(* IEC 61131-3 sources: PortalRobot/Portal_robot/Device/application/GVL, 22 files *)

(* ---- GVL_ALARM.gvl.st ---- *)
{attribute 'qualified_only'}
VAR_GLOBAL
	Command : ST_ALARM_COMMAND; // Команды управления журналом аварий
	Status  : ST_ALARM_STATUS; // Сводный статус аварий и предупреждений
	Events  : ARRAY [1..100] OF ST_ALARM_EVENT; // Кольцевой журнал событий
END_VAR

(* ---- GVL_AXIS.gvl.st ---- *)
{attribute 'qualified_only'}
VAR_GLOBAL
	arrAxis : ARRAY [1..3] OF ST_AXIS; // Команды, статусы и диагностика осей X, Y, Z
END_VAR

(* ---- GVL_AXIS_GROUP.gvl.st ---- *)
{attribute 'qualified_only'}
VAR_GLOBAL
	AxisGroup : ST_AXIS_GROUP; // Команды, статусы и диагностика группы XYZ
END_VAR

(* ---- GVL_CELL_CONTROL.gvl.st ---- *)
{attribute 'qualified_only'}
VAR_GLOBAL
	xGlobalError : BOOL; // Глобальная ошибка ячейки
	xReset       : BOOL; // Общий сброс ошибок ячейки
	xManual      : BOOL; // Ручной режим управления ячейкой
	xEnable      : BOOL; // Импульс включения оборудования ячейки
	xDisable     : BOOL; // Импульс отключения оборудования ячейки
	xStart       : BOOL; // Импульс запуска цикла или отмены ожидающей остановки
	xStop        : BOOL; // Импульс остановки автоматического цикла
END_VAR

(* ---- GVL_CELL_MANAGER.gvl.st ---- *)
{attribute 'qualified_only'}
VAR_GLOBAL
	Command : ST_CELL_COMMAND; // Команды менеджера ячейки
	Status  : ST_CELL_STATUS; // Рабочие статусы ячейки
	Diag    : ST_CELL_DIAG; // Состояние автомата ячейки
	Error   : ST_CELL_ERRORS; // Ошибки менеджера ячейки
END_VAR

(* ---- GVL_CELL_SAFETY_IO.gvl.st ---- *)
{attribute 'qualified_only'}
VAR_GLOBAL
	// Логические точки для назначения в Device I/O Mapping. Полярность НЗ-контактов
	// нормализуется при привязке: здесь TRUE всегда означает указанное состояние.
	// Начальное состояние стенда: двери закрыты, грибки отжаты, реле в норме.
	axDoorLockClosedInput : ARRAY [1..4] OF BOOL := [TRUE, TRUE, TRUE, TRUE];
	axDoorUnlockButtonInput : ARRAY [1..4] OF BOOL := [FALSE, FALSE, FALSE, FALSE];
	axEmergencyStopButtonStationInput : ARRAY [1..4] OF BOOL := [FALSE, FALSE, FALSE, FALSE];
	axEmergencyStopCabinetInput : ARRAY [1..2] OF BOOL := [FALSE, FALSE];
	xEmergencyStopMpgInput : BOOL := FALSE;
	xPhaseRelayOkInput    : BOOL := TRUE;
	xPressureRelayOkInput : BOOL := TRUE;
	xSafetyRelayOkInput   : BOOL := TRUE;
	xCellStartButtonInput : BOOL := FALSE;
	xCellStopButtonInput  : BOOL := FALSE;
	xCellResetButtonInput : BOOL := FALSE;
	xMpgAxisXInput : BOOL := FALSE;
	xMpgAxisYInput : BOOL := FALSE;
	xMpgAxisZInput : BOOL := FALSE;
	xMpgMultiplier1Input : BOOL := FALSE;
	xMpgMultiplier10Input : BOOL := FALSE;
	xMpgMultiplier100Input : BOOL := FALSE;

	// Выходы для назначения на физические каналы.
	axDoorUnlockOutput : ARRAY [1..4] OF BOOL;
	axDoorButtonLampOutput : ARRAY [1..4] OF BOOL;
	xSafetyRelayResetOutput : BOOL;
	// Светосигнальная колонна: готовые уровни с миганием из PLC_PRG.RunSignalTower.
	xSignalTowerRedOutput   : BOOL;
	xSignalTowerAmberOutput : BOOL;
	xSignalTowerGreenOutput : BOOL;
END_VAR

(* ---- GVL_CELL_SETTINGS.gvl.st ---- *)
{attribute 'qualified_only'}
VAR_GLOBAL CONSTANT
	// Максимальное число слотов магазина, используемое в статических границах массивов.
	NumberDetail : SINT := 70; // Максимальное число слотов магазина
END_VAR

VAR_GLOBAL
	//Порядок команд для смены, загрузки и выгрузки станков
	CHANGE_MACHINE : ARRAY [0..40] OF ST_MACHINE_RECIPE // Рецепт смены детали в станке
	:=[
	   (eCommand := E_MACHINE_STATE.DOOR_OPEN),
	   (eCommand := E_MACHINE_STATE.ROBOT_ACTION, eRobotAction := E_ROBOT_ACTION.ROTATE_TO_DETAIL),
	   (eCommand := E_MACHINE_STATE.ROBOT_ACTION, eRobotAction := E_ROBOT_ACTION.UNCLAMP_2),
	   (eCommand := E_MACHINE_STATE.ROBOT_MOVE, stPoint := E_MACHINE_POINTS.CHUCK_APPROACH),
	   (eCommand := E_MACHINE_STATE.ROBOT_MOVE, stPoint := E_MACHINE_POINTS.CHUCK),
	   (eCommand := E_MACHINE_STATE.ROBOT_ACTION, eRobotAction := E_ROBOT_ACTION.CLAMP_2),
	   (eCommand := E_MACHINE_STATE.CHUCK_OPEN),
	   (eCommand := E_MACHINE_STATE.ROBOT_MOVE, stPoint := E_MACHINE_POINTS.CHUCK_APPROACH),
	   (eCommand := E_MACHINE_STATE.ROBOT_ACTION, eRobotAction := E_ROBOT_ACTION.ROTATE_TO_BLANK),
	   (eCommand := E_MACHINE_STATE.ROBOT_MOVE, stPoint := E_MACHINE_POINTS.CHUCK),
	   (eCommand := E_MACHINE_STATE.CHUCK_CLOSE),
	   (eCommand := E_MACHINE_STATE.ROBOT_ACTION, eRobotAction := E_ROBOT_ACTION.UNCLAMP_1),
	   (eCommand := E_MACHINE_STATE.ROBOT_MOVE, stPoint := E_MACHINE_POINTS.CHUCK_APPROACH),
	   (eCommand := E_MACHINE_STATE.ROBOT_MOVE, stPoint := E_MACHINE_POINTS.ABOVE, xRobotDone := TRUE),
	   (eCommand := E_MACHINE_STATE.DOOR_CLOSE),
	   (eCommand := E_MACHINE_STATE.CYCLE_START),
	   (eCommand := E_MACHINE_STATE.DONE)

];
	LOAD_MACHINE : ARRAY [0..40] OF ST_MACHINE_RECIPE // Рецепт загрузки станка
	:=[
	   (eCommand := E_MACHINE_STATE.DOOR_OPEN),
	   (eCommand := E_MACHINE_STATE.ROBOT_ACTION, eRobotAction := E_ROBOT_ACTION.ROTATE_TO_BLANK),
	   (eCommand := E_MACHINE_STATE.ROBOT_MOVE, stPoint := E_MACHINE_POINTS.CHUCK_APPROACH),
	   (eCommand := E_MACHINE_STATE.ROBOT_MOVE, stPoint := E_MACHINE_POINTS.CHUCK),
	   (eCommand := E_MACHINE_STATE.CHUCK_CLOSE),
	   (eCommand := E_MACHINE_STATE.ROBOT_ACTION, eRobotAction := E_ROBOT_ACTION.UNCLAMP_1),
	   (eCommand := E_MACHINE_STATE.ROBOT_MOVE, stPoint := E_MACHINE_POINTS.CHUCK_APPROACH),
	   (eCommand := E_MACHINE_STATE.ROBOT_MOVE, stPoint := E_MACHINE_POINTS.ABOVE, xRobotDone := TRUE),
	   (eCommand := E_MACHINE_STATE.DOOR_CLOSE),
	   (eCommand := E_MACHINE_STATE.CYCLE_START),
	   (eCommand := E_MACHINE_STATE.DONE)
	];

	UNLOAD_MACHINE : ARRAY [0..40] OF ST_MACHINE_RECIPE // Рецепт выгрузки станка
	:=[
	   (eCommand := E_MACHINE_STATE.DOOR_OPEN),
	   (eCommand := E_MACHINE_STATE.ROBOT_ACTION, eRobotAction := E_ROBOT_ACTION.ROTATE_TO_DETAIL),
	   (eCommand := E_MACHINE_STATE.ROBOT_ACTION, eRobotAction := E_ROBOT_ACTION.UNCLAMP_2),
	   (eCommand := E_MACHINE_STATE.ROBOT_MOVE, stPoint := E_MACHINE_POINTS.CHUCK_APPROACH),
	   (eCommand := E_MACHINE_STATE.ROBOT_MOVE, stPoint := E_MACHINE_POINTS.CHUCK),
	   (eCommand := E_MACHINE_STATE.ROBOT_ACTION, eRobotAction := E_ROBOT_ACTION.CLAMP_2),
	   (eCommand := E_MACHINE_STATE.CHUCK_OPEN),
	   (eCommand := E_MACHINE_STATE.ROBOT_MOVE, stPoint := E_MACHINE_POINTS.CHUCK_APPROACH),
	   (eCommand := E_MACHINE_STATE.ROBOT_MOVE, stPoint := E_MACHINE_POINTS.ABOVE, xRobotDone := TRUE),
	   (eCommand := E_MACHINE_STATE.DOOR_CLOSE),
	   (eCommand := E_MACHINE_STATE.DONE)
	];
END_VAR

(* ---- GVL_DETAIL.gvl.st ---- *)
{attribute 'qualified_only'}
VAR_GLOBAL
	arrDetail : ARRAY [1..GVL_CELL_SETTINGS.NumberDetail] OF ST_DETAIL; // Содержимое слотов магазина
END_VAR

(* ---- GVL_HMI.gvl.st ---- *)
{attribute 'qualified_only'}
VAR_GLOBAL
	// Команды и настройки, получаемые от HMI.
	xCellEnable       : BOOL; // Импульс включения оборудования ячейки
	xCellDisable      : BOOL; // Импульс отключения оборудования ячейки
	xCellStart        : BOOL; // Импульс запуска автоматического цикла
	xCellStop         : BOOL; // Импульс остановки автоматического цикла
	xCellReset        : BOOL; // Общий сброс ошибок ячейки
	xAlarmResetWarnings : BOOL; // Импульс сброса накопленных предупреждений
	xCellManual       : BOOL; // Ручной режим управления ячейкой
	lrOffsetX          : LREAL; // Ручное смещение по оси X
	lrOffsetY          : LREAL; // Ручное смещение по оси Y
	lrOffsetZ          : LREAL; // Ручное смещение по оси Z
	xModbusMode        : BOOL; // TRUE: внешний робот по Modbus
	xRobotDrivesEnable : BOOL; // Импульс включения приводов робота
	xRobotDrivesDisable: BOOL; // Импульс отключения приводов робота
	xRobotStop         : BOOL; // Импульс контролируемой остановки робота
	xRobotReset        : BOOL; // Импульс сброса ошибок робота и приводов
	xMagazineEnable    : BOOL; // Импульс включения магазина
	xMagazineDisable   : BOOL; // Импульс отключения магазина
	xMagazineFillBlanks: BOOL; // Заполнить активные слоты магазина заготовками
	xMagazineClear     : BOOL; // Полностью очистить магазин
	{attribute 'symbol' := 'readwrite'}
	xMagazineCycleSlot : BOOL; // Переключить содержимое выбранного слота
	{attribute 'symbol' := 'readwrite'}
	uiMagazineEditSlot : UINT; // Номер слота, изменяемого оператором
	axMachineEnable    : ARRAY [1..3] OF BOOL; // Импульсы включения отдельных станков
	axMachineDisable   : ARRAY [1..3] OF BOOL; // Импульсы отключения отдельных станков
	axMachineReset     : ARRAY [1..3] OF BOOL; // Команды сброса ошибок отдельных станков
	{attribute 'symbol' := 'readwrite'}
	axMachineSetBlank  : ARRAY [1..3] OF BOOL; // Подтвердить заготовку в патроне
	{attribute 'symbol' := 'readwrite'}
	axMachineSetDetail : ARRAY [1..3] OF BOOL; // Подтвердить готовую деталь в патроне
	{attribute 'symbol' := 'readwrite'}
	axMachineAcceptDoor: ARRAY [1..3] OF BOOL; // Подтвердить закрытие двери
	{attribute 'symbol' := 'readwrite'}
	axMachineRejectDoor: ARRAY [1..3] OF BOOL; // Отказаться от закрытия двери
	{attribute 'symbol' := 'readwrite'}
	axMachineAcceptRun : ARRAY [1..3] OF BOOL; // Подтвердить запуск обработки
	{attribute 'symbol' := 'readwrite'}
	axMachineRejectRun : ARRAY [1..3] OF BOOL; // Отказаться от запуска обработки
	axMachineUsed      : ARRAY [1..3] OF BOOL := [TRUE, TRUE, TRUE]; // Станки в автоматической работе
	xUseHmiCycleTime   : ARRAY [1..3] OF BOOL := [TRUE, TRUE, TRUE]; // Использовать заданное время цикла
	tMachineCycleTime  : ARRAY [1..3] OF TIME := [T#60S, T#60S, T#60S]; // Время цикла станков
	{attribute 'symbol' := 'readwrite'}
	MagazineRows       : UINT := 7; // Число строк магазина
	{attribute 'symbol' := 'readwrite'}
	MagazineColumns    : UINT := 10; // Число столбцов магазина
	{attribute 'symbol' := 'readwrite'}
	MagazinePitchX     : LREAL := 80.0; // Шаг слотов по оси X
	{attribute 'symbol' := 'readwrite'}
	MagazinePitchY     : LREAL := 190.0; // Шаг слотов по оси Y
	{attribute 'symbol' := 'readwrite'}
	MagazineSafeZ_1    : LREAL := 0.0; // Безопасная высота над магазином
	{attribute 'symbol' := 'readwrite'}
	MagazineSafeZ_2    : LREAL := 1400.0; // Безопасная высота внутри магазина при смене
	stRobotCommand     : ST_ROBOT_COMMAND; // Ручная команда роботу или магазину

	// Данные, передаваемые в HMI.
	udiPlcHeartbeat : UDINT; // Счётчик циклов PLC для контроля связи
	xGlobalError    : BOOL; // Активна общая ошибка ячейки
	lrActualX       : LREAL; // Текущая координата X
	lrActualY       : LREAL; // Текущая координата Y
	lrActualZ       : LREAL; // Текущая координата Z

	stCellStatus : ST_CELL_STATUS; // Рабочее состояние автоматического цикла
	stCellDiag   : ST_CELL_DIAG; // Текущий шаг менеджера ячейки
	stCellError  : ST_CELL_ERRORS; // Активные и последние ошибки менеджера ячейки

	stRobotStatus : ST_ROBOT_STATUS; // Состояние робота и двух захватов
	stRobotDiag   : ST_ROBOT_DIAG; // Текущее действие и целевая точка робота
	stRobotError  : ST_ROBOT_ERRORS; // Активные и последние ошибки робота

	{attribute 'symbol' := 'read'}
	astMachineStatus   : ARRAY [1..3] OF ST_MACHINE_PUBLIC; // Рабочие состояния станков
	astMachineIoStatus : ARRAY [1..3] OF ST_MACHINE_IO_STATUS; // Двери, патроны и циклы станков
	astMachineDiag     : ARRAY [1..3] OF ST_MACHINE_DIAG; // Текущие шаги и операции станков
	astMachineError    : ARRAY [1..3] OF ST_MACHINE_ERRORS; // Активные и последние ошибки станков

	{attribute 'symbol' := 'read'}
	stMagazineStatus : ST_MAGAZINE_STATUS; // Готовность и текущая операция магазина
	stMagazineDiag   : ST_MAGAZINE_DIAG; // Текущий шаг магазина
	stMagazineError  : ST_MAGAZINE_ERRORS; // Активные и последние ошибки магазина
	astMagazineSlot  : ARRAY [1..GVL_CELL_SETTINGS.NumberDetail] OF ST_DETAIL; // Содержимое слотов магазина
	stAlarmStatus : ST_ALARM_STATUS; // Сводный статус аварий и предупреждений
	astAlarmEvent : ARRAY [1..100] OF ST_ALARM_EVENT; // Журнал активных и зафиксированных событий

	// Совместимость с существующей визуализацией до штатного обновления XML.
	HMI : ST_HMI; // Старый путь GVL_HMI.HMI.ActualX/Y/Z
END_VAR

(* ---- GVL_MACHINE.gvl.st ---- *)
{attribute 'qualified_only'}
VAR_GLOBAL
	Command    : ARRAY [1..3] OF ST_MACHINE_COMMAND; // Команды станков и робота
	Status     : ARRAY [1..3] OF ST_MACHINE_PUBLIC; // Рабочие статусы станков
	Diag       : ARRAY [1..3] OF ST_MACHINE_DIAG; // Состояния автоматов станков
	Error      : ARRAY [1..3] OF ST_MACHINE_ERRORS; // Ошибки станков
END_VAR

(* ---- GVL_MAGAZINE.gvl.st ---- *)
{attribute 'qualified_only'}
VAR_GLOBAL
	astPartStatus : ARRAY [1..2] OF ST_MAGAZINE_STATUS; // Статус только операций робота, без механического обмена
	astAutoCommand : ARRAY [1..GVL_CELL_SETTINGS.MagazineCount] OF ST_MAGAZINE_COMMAND;
	astCommand : ARRAY [1..GVL_CELL_SETTINGS.MagazineCount] OF ST_ROBOT_COMMAND;
	astStatus : ARRAY [1..GVL_CELL_SETTINGS.MagazineCount] OF ST_MAGAZINE_STATUS;
	astDiag : ARRAY [1..GVL_CELL_SETTINGS.MagazineCount] OF ST_MAGAZINE_DIAG;
	astError : ARRAY [1..GVL_CELL_SETTINGS.MagazineCount] OF ST_MAGAZINE_ERRORS;
END_VAR

(* ---- GVL_MAGAZINE_AXIS.gvl.st ---- *)
{attribute 'qualified_only'}
VAR_GLOBAL
	// Legacy-объявление оставлено до удаления SoftMotion-узлов Magazine_1/2 через
	// CODESYS. Активная программа массив не читает, не пишет и FB_AXIS для него не создаёт.
	astAxis : ARRAY [1..GVL_CELL_SETTINGS.MagazineCount] OF ST_AXIS;
END_VAR

(* ---- GVL_MOTION_MANAGER.gvl.st ---- *)
{attribute 'qualified_only'}
VAR_GLOBAL
	stMotionManager: ST_MOTION_MANAGER;
END_VAR

(* ---- GVL_MULTI_TYPE.gvl.st ---- *)
{attribute 'qualified_only'}
VAR_GLOBAL
	Config       : ST_MULTI_TYPE_CONFIG; // Активная конфигурация типов продукции
	ConfigStatus : ST_MULTI_TYPE_CONFIG_STATUS; // Разрешения редактирования конфигурации
	CycleStatus  : ST_CELL_CYCLE_STATUS; // Диагностика универсального автомата ячейки
END_VAR

(* ---- GVL_POINT.gvl.st ---- *)
{attribute 'qualified_only'}
VAR_GLOBAL
	Points : ARRAY [0..iPointNumber] OF ST_POINT; // Глобальная таблица именованных точек
END_VAR

VAR_GLOBAL PERSISTENT RETAIN
	// Постоянное хранилище базовых точек в энергонезависимой памяти контроллера.
	// Размер 15 сохранён ради совместимости со старой раскладкой: позиции 2, 6 и 10
	// (legacy MACHINE_x_INSIDE) больше не публикуются и не участвуют в готовности.
	astRetainPoints : ARRAY [1..iPersistentPointCapacity] OF ST_POINT;
	udiPointStorageVersion : UDINT;
END_VAR

VAR_GLOBAL CONSTANT
	iPointNumber : INT := 100; // Максимальный индекс таблицы точек
	iEditablePointCount : INT := 12;
	iPersistentPointCapacity : INT := 15;
	udiExpectedPointStorageVersion : UDINT := UDINT#1;
END_VAR

(* ---- GVL_POINT_MANAGER.gvl.st ---- *)
{attribute 'qualified_only'}
VAR_GLOBAL
	PointManager : ST_POINT_MANAGER; // Команды, статусы и диагностика проверки точки
END_VAR

(* ---- GVL_ROBOT.gvl.st ---- *)
{attribute 'qualified_only'}
VAR_GLOBAL
	Command       : ST_ROBOT_COMMAND; // Выбранная команда робота
	ModbusCommand : ST_ROBOT_COMMAND; // Команда внешнему роботу
	Status        : ST_ROBOT_STATUS; // Рабочие статусы робота
	Diag          : ST_ROBOT_DIAG; // Состояние автомата робота
	Error         : ST_ROBOT_ERRORS; // Активные и последние ошибки робота
	GripperDiag   : ST_GRIPPER_DIAG; // Диагностика внутреннего блока захвата
	GripperError  : ST_GRIPPER_ERRORS; // Активные и последние ошибки захвата

	xModbusBusy  : BOOL; // Внешний робот выполняет команду
	xModbusDone  : BOOL; // Внешний робот завершил команду
	xModbusError : BOOL; // Ошибка внешнего робота или обмена
END_VAR

(* ---- GVL_ROBOT_MODBUS.gvl.st ---- *)
{attribute 'qualified_only'}
VAR_GLOBAL
	xModeActive             : BOOL; // TRUE, когда применён MODBUS_TCP
	xRobotModeChangeAllowed : BOOL; // Авторитетное разрешение PLC
	xSettingsChangeAllowed  : BOOL; // Авторитетное разрешение PLC
	xReconnectRequest       : BOOL; // Одноцикловый запрос переподключения клиента
	Config                  : ST_ROBOT_MODBUS_CONFIG;
	Status                  : ST_ROBOT_MODBUS_STATUS;
	Command                 : ST_ROBOT_COMMAND;
	auiWriteRegisters       : ARRAY [0..8] OF UINT; // 1001..1009
	auiReadRegisters        : ARRAY [0..16] OF UINT; // 1101..1117
END_VAR

(* ---- GVL_ROBOT_MODBUS_RETAIN.gvl.st ---- *)
{attribute 'qualified_only'}
VAR_GLOBAL RETAIN
	eControlMode      : E_ROBOT_CONTROL_MODE := E_ROBOT_CONTROL_MODE.SOFTMOTION;
	aIpAddress        : ARRAY [0..3] OF BYTE := [BYTE#0, BYTE#0, BYTE#0, BYTE#0];
	uiPort            : UINT := UINT#502;
	uiUnitId          : UINT := UINT#1;
	tResponseTimeout  : TIME := T#500MS;
	tPollInterval     : TIME := T#50MS;
	tHeartbeatTimeout : TIME := T#2S;
	tCommandStartTimeout : TIME := T#30S;
	tCommandTimeout   : TIME := T#600S;
END_VAR

(* ---- GVL_STATISTIC.gvl.st ---- *)
{attribute 'qualified_only'}
VAR_GLOBAL
	stStatistic			: ST_STATISTIC;
END_VAR

(* ---- GVL_TEST_IO.gvl.st ---- *)
{attribute 'qualified_only'}
VAR_GLOBAL
	// Логический вход. Физический адрес назначается отдельно в Device I/O Mapping CODESYS.
	xSc500BenchKeyInput : BOOL := FALSE;
END_VAR

(* ---- GVL_TWO_PALLET.gvl.st ---- *)
{attribute 'qualified_only'}
VAR_GLOBAL
	Axis1 : REFERENCE TO AXIS_REF_SM3; // Каждый скан REF= Magazine_1 в RunTwoPalletAxis
	Axis2 : REFERENCE TO AXIS_REF_SM3; // Каждый скан REF= Magazine_2 в RunTwoPalletAxis
	astAxis : ARRAY [1..2] OF ST_AXIS;
	astInput : ARRAY [1..2] OF ST_TWO_PALLET_INPUT; // Физические входы: НЕ записываются из HMI
	astOutput : ARRAY [1..2] OF ST_TWO_PALLET_OUTPUT;
	astSimulationConfig : ARRAY [1..2] OF ST_TWO_PALLET_CONFIG; // Только виртуальная среда; не RETAIN
	astActiveConfig : ARRAY [1..2] OF ST_TWO_PALLET_CONFIG; // Конфигурация текущей среды
	astStatus : ARRAY [1..2] OF ST_TWO_PALLET_STATUS;
	astDiag : ARRAY [1..2] OF ST_TWO_PALLET_DIAG;
	astError : ARRAY [1..2] OF ST_TWO_PALLET_ERRORS;
	auiCommand : ARRAY [1..2] OF UINT;
	auiValue : ARRAY [1..2] OF UINT;
	audiRevision : ARRAY [1..2] OF UDINT;
	xModeChangeAllowed : BOOL;
	xModeChanged : BOOL;
	astStatic : ARRAY [1..2] OF ST_MAGAZINE_INVENTORY;
	axSimulationAutoSwapEnabled : ARRAY [1..2] OF BOOL; // Только виртуальная среда; не RETAIN
END_VAR
VAR_GLOBAL RETAIN
	uiMode : UINT := UINT#1; // По умолчанию два двухпалетных; 0: два статичных; 1: два двухпалетных
	astConfig : ARRAY [1..2] OF ST_TWO_PALLET_CONFIG;
	astStore : ARRAY [1..2] OF ST_TWO_PALLET_STORE;
	lrStaticPitchX : LREAL := 60.0;
	lrStaticPitchY : LREAL := 60.0;
	lrTwinPitchX : LREAL := 70.0;
	lrTwinPitchY : LREAL := 70.0;
	axAutoSwapEnabled : ARRAY [1..2] OF BOOL := [TRUE, TRUE];
	xAutoSwapDefaultsApplied : BOOL; // Однократная инициализация новой RETAIN-настройки
END_VAR
